        ! Point 20: (1430, 300) [work]
        CurrentX:=1430;
        CurrentY:=300;
        pCurrent.trans:=[-1*CurrentX,CurrentY,WorkZ];
        pCurrent.rot:=OrientZYX(0,0,180);
        pCurrent.robconf:=[1,0,-2,0];
        CalcTrack:=Bed1Wyong.uframe.trans.x+pCurrent.trans.x;
        IF CurrentY<1000 THEN CalcTrack:=CalcTrack+1200; ENDIF
        IF CalcTrack<TrackMin THEN CalcTrack:=TrackMin; ENDIF
        IF CalcTrack>TrackMax THEN CalcTrack:=TrackMax; ENDIF
        pCurrent.extax:=[CalcTrack,9E+09,9E+09,9E+09,9E+09,9E+09];
        MoveL pCurrent,vTravel,fine,tHeli\WObj:=Bed1Wyong;

        ! Point 21: (1730, 300) [work]
        CurrentX:=1730;
        CurrentY:=300;
        pCurrent.trans:=[-1*CurrentX,CurrentY,WorkZ];
        pCurrent.rot:=OrientZYX(0,0,180);
        pCurrent.robconf:=[1,0,-2,0];
        CalcTrack:=Bed1Wyong.uframe.trans.x+pCurrent.trans.x;
        IF CurrentY<1000 THEN CalcTrack:=CalcTrack+1200; ENDIF
        IF CalcTrack<TrackMin THEN CalcTrack:=TrackMin; ENDIF
        IF CalcTrack>TrackMax THEN CalcTrack:=TrackMax; ENDIF
        pCurrent.extax:=[CalcTrack,9E+09,9E+09,9E+09,9E+09,9E+09];
        MoveL pCurrent,vTravel,fine,tHeli\WObj:=Bed1Wyong;

        ! Point 22: (1730, 1550) [work]
        CurrentX:=1730;
        CurrentY:=1550;
        pCurrent.trans:=[-1*CurrentX,CurrentY,WorkZ];
        pCurrent.rot:=OrientZYX(0,0,180);
        pCurrent.robconf:=[1,0,-2,0];
        CalcTrack:=Bed1Wyong.uframe.trans.x+pCurrent.trans.x;
        IF CurrentY<1000 THEN CalcTrack:=CalcTrack+1200; ENDIF
        IF CalcTrack<TrackMin THEN CalcTrack:=TrackMin; ENDIF
        IF CalcTrack>TrackMax THEN CalcTrack:=TrackMax; ENDIF
        pCurrent.extax:=[CalcTrack,9E+09,9E+09,9E+09,9E+09,9E+09];
        MoveL pCurrent,vTravel,fine,tHeli\WObj:=Bed1Wyong;

        ! Point 23: (2030, 1550) [work]
        CurrentX:=2030;
        CurrentY:=1550;
        pCurrent.trans:=[-1*CurrentX,CurrentY,WorkZ];
        pCurrent.rot:=OrientZYX(0,0,180);
        pCurrent.robconf:=[1,0,-2,0];
        CalcTrack:=Bed1Wyong.uframe.trans.x+pCurrent.trans.x;
        IF CurrentY<1000 THEN CalcTrack:=CalcTrack+1200; ENDIF
        IF CalcTrack<TrackMin THEN CalcTrack:=TrackMin; ENDIF
        IF CalcTrack>TrackMax THEN CalcTrack:=TrackMax; ENDIF
        pCurrent.extax:=[CalcTrack,9E+09,9E+09,9E+09,9E+09,9E+09];
        MoveL pCurrent,vTravel,fine,tHeli\WObj:=Bed1Wyong;

        ! Point 24: (2030, 300) [work]
        CurrentX:=2030;
        CurrentY:=300;
        pCurrent.trans:=[-1*CurrentX,CurrentY,WorkZ];
        pCurrent.rot:=OrientZYX(0,0,180);
        pCurrent.robconf:=[1,0,-2,0];
        CalcTrack:=Bed1Wyong.uframe.trans.x+pCurrent.trans.x;
        IF CurrentY<1000 THEN CalcTrack:=CalcTrack+1200; ENDIF
        IF CalcTrack<TrackMin THEN CalcTrack:=TrackMin; ENDIF
        IF CalcTrack>TrackMax THEN CalcTrack:=TrackMax; ENDIF
        pCurrent.extax:=[CalcTrack,9E+09,9E+09,9E+09,9E+09,9E+09];
        MoveL pCurrent,vTravel,fine,tHeli\WObj:=Bed1Wyong;

        ! Point 25: (2330, 300) [work]
        CurrentX:=2330;
        CurrentY:=300;
        pCurrent.trans:=[-1*CurrentX,CurrentY,WorkZ];
        pCurrent.rot:=OrientZYX(0,0,180);
        pCurrent.robconf:=[1,0,-2,0];
        CalcTrack:=Bed1Wyong.uframe.trans.x+pCurrent.trans.x;
        IF CurrentY<1000 THEN CalcTrack:=CalcTrack+1200; ENDIF
        IF CalcTrack<TrackMin THEN CalcTrack:=TrackMin; ENDIF
        IF CalcTrack>TrackMax THEN CalcTrack:=TrackMax; ENDIF
        pCurrent.extax:=[CalcTrack,9E+09,9E+09,9E+09,9E+09,9E+09];
        MoveL pCurrent,vTravel,fine,tHeli\WObj:=Bed1Wyong;

        ! Point 26: (2330, 1550) [work]
        CurrentX:=2330;
        CurrentY:=1550;
        pCurrent.trans:=[-1*CurrentX,CurrentY,WorkZ];
        pCurrent.rot:=OrientZYX(0,0,180);
        pCurrent.robconf:=[1,0,-2,0];
        CalcTrack:=Bed1Wyong.uframe.trans.x+pCurrent.trans.x;
        IF CurrentY<1000 THEN CalcTrack:=CalcTrack+1200; ENDIF
        IF CalcTrack<TrackMin THEN CalcTrack:=TrackMin; ENDIF
        IF CalcTrack>TrackMax THEN CalcTrack:=TrackMax; ENDIF
        pCurrent.extax:=[CalcTrack,9E+09,9E+09,9E+09,9E+09,9E+09];
        MoveL pCurrent,vTravel,fine,tHeli\WObj:=Bed1Wyong;

        ! Point 27: (2630, 1550) [work]
        CurrentX:=2630;
        CurrentY:=1550;
        pCurrent.trans:=[-1*CurrentX,CurrentY,WorkZ];
        pCurrent.rot:=OrientZYX(0,0,180);
        pCurrent.robconf:=[1,0,-2,0];
        CalcTrack:=Bed1Wyong.uframe.trans.x+pCurrent.trans.x;
        IF CurrentY<1000 THEN CalcTrack:=CalcTrack+1200; ENDIF
        IF CalcTrack<TrackMin THEN CalcTrack:=TrackMin; ENDIF
        IF CalcTrack>TrackMax THEN CalcTrack:=TrackMax; ENDIF
        pCurrent.extax:=[CalcTrack,9E+09,9E+09,9E+09,9E+09,9E+09];
        MoveL pCurrent,vTravel,fine,tHeli\WObj:=Bed1Wyong;

        ! Point 28: (2630, 300) [work]
        CurrentX:=2630;
        CurrentY:=300;
        pCurrent.trans:=[-1*CurrentX,CurrentY,WorkZ];
        pCurrent.rot:=OrientZYX(0,0,180);
        pCurrent.robconf:=[1,0,-2,0];
        CalcTrack:=Bed1Wyong.uframe.trans.x+pCurrent.trans.x;
        IF CurrentY<1000 THEN CalcTrack:=CalcTrack+1200; ENDIF
        IF CalcTrack<TrackMin THEN CalcTrack:=TrackMin; ENDIF
        IF CalcTrack>TrackMax THEN CalcTrack:=TrackMax; ENDIF
        pCurrent.extax:=[CalcTrack,9E+09,9E+09,9E+09,9E+09,9E+09];
        MoveL pCurrent,vTravel,fine,tHeli\WObj:=Bed1Wyong;

        ! Point 29: (2930, 300) [work]
        CurrentX:=2930;
        CurrentY:=300;
        pCurrent.trans:=[-1*CurrentX,CurrentY,WorkZ];
        pCurrent.rot:=OrientZYX(0,0,180);
        pCurrent.robconf:=[1,0,-2,0];
        CalcTrack:=Bed1Wyong.uframe.trans.x+pCurrent.trans.x;
        IF CurrentY<1000 THEN CalcTrack:=CalcTrack+1200; ENDIF
        IF CalcTrack<TrackMin THEN CalcTrack:=TrackMin; ENDIF
        IF CalcTrack>TrackMax THEN CalcTrack:=TrackMax; ENDIF
        pCurrent.extax:=[CalcTrack,9E+09,9E+09,9E+09,9E+09,9E+09];
        MoveL pCurrent,vTravel,fine,tHeli\WObj:=Bed1Wyong;

        ! Point 30: (2930, 1550) [work]
        CurrentX:=2930;
        CurrentY:=1550;
        pCurrent.trans:=[-1*CurrentX,CurrentY,WorkZ];
        pCurrent.rot:=OrientZYX(0,0,180);
        pCurrent.robconf:=[1,0,-2,0];
        CalcTrack:=Bed1Wyong.uframe.trans.x+pCurrent.trans.x;
        IF CurrentY<1000 THEN CalcTrack:=CalcTrack+1200; ENDIF
        IF CalcTrack<TrackMin THEN CalcTrack:=TrackMin; ENDIF
        IF CalcTrack>TrackMax THEN CalcTrack:=TrackMax; ENDIF
        pCurrent.extax:=[CalcTrack,9E+09,9E+09,9E+09,9E+09,9E+09];
        MoveL pCurrent,vTravel,fine,tHeli\WObj:=Bed1Wyong;

        ! Point 31: (3230, 1550) [work]
        CurrentX:=3230;
        CurrentY:=1550;
        pCurrent.trans:=[-1*CurrentX,CurrentY,WorkZ];
        pCurrent.rot:=OrientZYX(0,0,180);
        pCurrent.robconf:=[1,0,-2,0];
        CalcTrack:=Bed1Wyong.uframe.trans.x+pCurrent.trans.x;
        IF CurrentY<1000 THEN CalcTrack:=CalcTrack+1200; ENDIF
        IF CalcTrack<TrackMin THEN CalcTrack:=TrackMin; ENDIF
        IF CalcTrack>TrackMax THEN CalcTrack:=TrackMax; ENDIF
        pCurrent.extax:=[CalcTrack,9E+09,9E+09,9E+09,9E+09,9E+09];
        MoveL pCurrent,vTravel,fine,tHeli\WObj:=Bed1Wyong;

        ! Point 32: (3230, 300) [work]
        CurrentX:=3230;
        CurrentY:=300;
        pCurrent.trans:=[-1*CurrentX,CurrentY,WorkZ];
        pCurrent.rot:=OrientZYX(0,0,180);
        pCurrent.robconf:=[1,0,-2,0];
        CalcTrack:=Bed1Wyong.uframe.trans.x+pCurrent.trans.x;
        IF CurrentY<1000 THEN CalcTrack:=CalcTrack+1200; ENDIF
        IF CalcTrack<TrackMin THEN CalcTrack:=TrackMin; ENDIF
        IF CalcTrack>TrackMax THEN CalcTrack:=TrackMax; ENDIF
        pCurrent.extax:=[CalcTrack,9E+09,9E+09,9E+09,9E+09,9E+09];
        MoveL pCurrent,vTravel,fine,tHeli\WObj:=Bed1Wyong;

        ! Point 33: (3530, 300) [work]
        CurrentX:=3530;
        CurrentY:=300;
        pCurrent.trans:=[-1*CurrentX,CurrentY,WorkZ];
        pCurrent.rot:=OrientZYX(0,0,180);
        pCurrent.robconf:=[1,0,-2,0];
        CalcTrack:=Bed1Wyong.uframe.trans.x+pCurrent.trans.x;
        IF CurrentY<1000 THEN CalcTrack:=CalcTrack+1200; ENDIF
        IF CalcTrack<TrackMin THEN CalcTrack:=TrackMin; ENDIF
        IF CalcTrack>TrackMax THEN CalcTrack:=TrackMax; ENDIF
        pCurrent.extax:=[CalcTrack,9E+09,9E+09,9E+09,9E+09,9E+09];
        MoveL pCurrent,vTravel,fine,tHeli\WObj:=Bed1Wyong;

        ! Point 34: (3530, 1550) [work]
        CurrentX:=3530;
        CurrentY:=1550;
        pCurrent.trans:=[-1*CurrentX,CurrentY,WorkZ];
        pCurrent.rot:=OrientZYX(0,0,180);
        pCurrent.robconf:=[1,0,-2,0];
        CalcTrack:=Bed1Wyong.uframe.trans.x+pCurrent.trans.x;
        IF CurrentY<1000 THEN CalcTrack:=CalcTrack+1200; ENDIF
        IF CalcTrack<TrackMin THEN CalcTrack:=TrackMin; ENDIF
        IF CalcTrack>TrackMax THEN CalcTrack:=TrackMax; ENDIF
        pCurrent.extax:=[CalcTrack,9E+09,9E+09,9E+09,9E+09,9E+09];
        MoveL pCurrent,vTravel,fine,tHeli\WObj:=Bed1Wyong;

        ! Point 35: (3830, 1550) [work]
        CurrentX:=3830;
        CurrentY:=1550;
        pCurrent.trans:=[-1*CurrentX,CurrentY,WorkZ];
        pCurrent.rot:=OrientZYX(0,0,180);
        pCurrent.robconf:=[1,0,-2,0];
        CalcTrack:=Bed1Wyong.uframe.trans.x+pCurrent.trans.x;
        IF CurrentY<1000 THEN CalcTrack:=CalcTrack+1200; ENDIF
        IF CalcTrack<TrackMin THEN CalcTrack:=TrackMin; ENDIF
        IF CalcTrack>TrackMax THEN CalcTrack:=TrackMax; ENDIF
        pCurrent.extax:=[CalcTrack,9E+09,9E+09,9E+09,9E+09,9E+09];
        MoveL pCurrent,vTravel,fine,tHeli\WObj:=Bed1Wyong;

        ! Point 36: (3830, 300) [work]
        CurrentX:=3830;
        CurrentY:=300;
        pCurrent.trans:=[-1*CurrentX,CurrentY,WorkZ];
        pCurrent.rot:=OrientZYX(0,0,180);
        pCurrent.robconf:=[1,0,-2,0];
        CalcTrack:=Bed1Wyong.uframe.trans.x+pCurrent.trans.x;
        IF CurrentY<1000 THEN CalcTrack:=CalcTrack+1200; ENDIF
        IF CalcTrack<TrackMin THEN CalcTrack:=TrackMin; ENDIF
        IF CalcTrack>TrackMax THEN CalcTrack:=TrackMax; ENDIF
        pCurrent.extax:=[CalcTrack,9E+09,9E+09,9E+09,9E+09,9E+09];
        MoveL pCurrent,vTravel,fine,tHeli\WObj:=Bed1Wyong;

        ! Point 37: (4130, 300) [work]
        CurrentX:=4130;
        CurrentY:=300;
        pCurrent.trans:=[-1*CurrentX,CurrentY,WorkZ];
        pCurrent.rot:=OrientZYX(0,0,180);
        pCurrent.robconf:=[1,0,-2,0];
        CalcTrack:=Bed1Wyong.uframe.trans.x+pCurrent.trans.x;
        IF CurrentY<1000 THEN CalcTrack:=CalcTrack+1200; ENDIF
        IF CalcTrack<TrackMin THEN CalcTrack:=TrackMin; ENDIF
        IF CalcTrack>TrackMax THEN CalcTrack:=TrackMax; ENDIF
        pCurrent.extax:=[CalcTrack,9E+09,9E+09,9E+09,9E+09,9E+09];
        MoveL pCurrent,vTravel,fine,tHeli\WObj:=Bed1Wyong;

        ! Point 38: (4130, 1550) [work]
        CurrentX:=4130;
        CurrentY:=1550;
        pCurrent.trans:=[-1*CurrentX,CurrentY,WorkZ];
        pCurrent.rot:=OrientZYX(0,0,180);
        pCurrent.robconf:=[1,0,-2,0];
        CalcTrack:=Bed1Wyong.uframe.trans.x+pCurrent.trans.x;
        IF CurrentY<1000 THEN CalcTrack:=CalcTrack+1200; ENDIF
        IF CalcTrack<TrackMin THEN CalcTrack:=TrackMin; ENDIF
        IF CalcTrack>TrackMax THEN CalcTrack:=TrackMax; ENDIF
        pCurrent.extax:=[CalcTrack,9E+09,9E+09,9E+09,9E+09,9E+09];
        MoveL pCurrent,vTravel,fine,tHeli\WObj:=Bed1Wyong;

        ! Point 39: (4430, 1550) [work]
        CurrentX:=4430;
        CurrentY:=1550;
        pCurrent.trans:=[-1*CurrentX,CurrentY,WorkZ];
        pCurrent.rot:=OrientZYX(0,0,180);
        pCurrent.robconf:=[1,0,-2,0];
        CalcTrack:=Bed1Wyong.uframe.trans.x+pCurrent.trans.x;
        IF CurrentY<1000 THEN CalcTrack:=CalcTrack+1200; ENDIF
        IF CalcTrack<TrackMin THEN CalcTrack:=TrackMin; ENDIF
        IF CalcTrack>TrackMax THEN CalcTrack:=TrackMax; ENDIF
        pCurrent.extax:=[CalcTrack,9E+09,9E+09,9E+09,9E+09,9E+09];
        MoveL pCurrent,vTravel,fine,tHeli\WObj:=Bed1Wyong;

        ! Point 40: (4430, 300) [work]
        CurrentX:=4430;
        CurrentY:=300;
        pCurrent.trans:=[-1*CurrentX,CurrentY,WorkZ];
        pCurrent.rot:=OrientZYX(0,0,180);
        pCurrent.robconf:=[1,0,-2,0];
        CalcTrack:=Bed1Wyong.uframe.trans.x+pCurrent.trans.x;
        IF CurrentY<1000 THEN CalcTrack:=CalcTrack+1200; ENDIF
        IF CalcTrack<TrackMin THEN CalcTrack:=TrackMin; ENDIF
        IF CalcTrack>TrackMax THEN CalcTrack:=TrackMax; ENDIF
        pCurrent.extax:=[CalcTrack,9E+09,9E+09,9E+09,9E+09,9E+09];
        MoveL pCurrent,vTravel,fine,tHeli\WObj:=Bed1Wyong;

        ! Point 41: (4730, 300) [work]
        CurrentX:=4730;
        CurrentY:=300;
        pCurrent.trans:=[-1*CurrentX,CurrentY,WorkZ];
        pCurrent.rot:=OrientZYX(0,0,180);
        pCurrent.robconf:=[1,0,-2,0];
        CalcTrack:=Bed1Wyong.uframe.trans.x+pCurrent.trans.x;
        IF CurrentY<1000 THEN CalcTrack:=CalcTrack+1200; ENDIF
        IF CalcTrack<TrackMin THEN CalcTrack:=TrackMin; ENDIF
        IF CalcTrack>TrackMax THEN CalcTrack:=TrackMax; ENDIF
        pCurrent.extax:=[CalcTrack,9E+09,9E+09,9E+09,9E+09,9E+09];
        MoveL pCurrent,vTravel,fine,tHeli\WObj:=Bed1Wyong;

        ! Point 42: (4730, 1550) [work]
        CurrentX:=4730;
        CurrentY:=1550;
        pCurrent.trans:=[-1*CurrentX,CurrentY,WorkZ];
        pCurrent.rot:=OrientZYX(0,0,180);
        pCurrent.robconf:=[1,0,-2,0];
        CalcTrack:=Bed1Wyong.uframe.trans.x+pCurrent.trans.x;
        IF CurrentY<1000 THEN CalcTrack:=CalcTrack+1200; ENDIF
        IF CalcTrack<TrackMin THEN CalcTrack:=TrackMin; ENDIF
        IF CalcTrack>TrackMax THEN CalcTrack:=TrackMax; ENDIF
        pCurrent.extax:=[CalcTrack,9E+09,9E+09,9E+09,9E+09,9E+09];
        MoveL pCurrent,vTravel,fine,tHeli\WObj:=Bed1Wyong;

        ! Point 43: (5030, 1550) [work]
        CurrentX:=5030;
        CurrentY:=1550;
        pCurrent.trans:=[-1*CurrentX,CurrentY,WorkZ];
        pCurrent.rot:=OrientZYX(0,0,180);
        pCurrent.robconf:=[1,0,-2,0];
        CalcTrack:=Bed1Wyong.uframe.trans.x+pCurrent.trans.x;
        IF CurrentY<1000 THEN CalcTrack:=CalcTrack+1200; ENDIF
        IF CalcTrack<TrackMin THEN CalcTrack:=TrackMin; ENDIF
        IF CalcTrack>TrackMax THEN CalcTrack:=TrackMax; ENDIF
        pCurrent.extax:=[CalcTrack,9E+09,9E+09,9E+09,9E+09,9E+09];
        MoveL pCurrent,vTravel,fine,tHeli\WObj:=Bed1Wyong;

        ! Point 44: (5030, 300) [work]
        CurrentX:=5030;
        CurrentY:=300;
        pCurrent.trans:=[-1*CurrentX,CurrentY,WorkZ];
        pCurrent.rot:=OrientZYX(0,0,180);
        pCurrent.robconf:=[1,0,-2,0];
        CalcTrack:=Bed1Wyong.uframe.trans.x+pCurrent.trans.x;
        IF CurrentY<1000 THEN CalcTrack:=CalcTrack+1200; ENDIF
        IF CalcTrack<TrackMin THEN CalcTrack:=TrackMin; ENDIF
        IF CalcTrack>TrackMax THEN CalcTrack:=TrackMax; ENDIF
        pCurrent.extax:=[CalcTrack,9E+09,9E+09,9E+09,9E+09,9E+09];
        MoveL pCurrent,vTravel,fine,tHeli\WObj:=Bed1Wyong;

        ! Point 45: (5330, 300) [work]
        CurrentX:=5330;
        CurrentY:=300;
        pCurrent.trans:=[-1*CurrentX,CurrentY,WorkZ];
        pCurrent.rot:=OrientZYX(0,0,180);
        pCurrent.robconf:=[1,0,-2,0];
        CalcTrack:=Bed1Wyong.uframe.trans.x+pCurrent.trans.x;
        IF CurrentY<1000 THEN CalcTrack:=CalcTrack+1200; ENDIF
        IF CalcTrack<TrackMin THEN CalcTrack:=TrackMin; ENDIF
        IF CalcTrack>TrackMax THEN CalcTrack:=TrackMax; ENDIF
        pCurrent.extax:=[CalcTrack,9E+09,9E+09,9E+09,9E+09,9E+09];
        MoveL pCurrent,vTravel,fine,tHeli\WObj:=Bed1Wyong;

        ! Point 46: (5330, 1550) [work]
        CurrentX:=5330;
        CurrentY:=1550;
        pCurrent.trans:=[-1*CurrentX,CurrentY,WorkZ];
        pCurrent.rot:=OrientZYX(0,0,180);
        pCurrent.robconf:=[1,0,-2,0];
        CalcTrack:=Bed1Wyong.uframe.trans.x+pCurrent.trans.x;
        IF CurrentY<1000 THEN CalcTrack:=CalcTrack+1200; ENDIF
        IF CalcTrack<TrackMin THEN CalcTrack:=TrackMin; ENDIF
        IF CalcTrack>TrackMax THEN CalcTrack:=TrackMax; ENDIF
        pCurrent.extax:=[CalcTrack,9E+09,9E+09,9E+09,9E+09,9E+09];
        MoveL pCurrent,vTravel,fine,tHeli\WObj:=Bed1Wyong;

        ! Point 47: (5630, 1550) [work]
        CurrentX:=5630;
        CurrentY:=1550;
        pCurrent.trans:=[-1*CurrentX,CurrentY,WorkZ];
        pCurrent.rot:=OrientZYX(0,0,180);
        pCurrent.robconf:=[1,0,-2,0];
        CalcTrack:=Bed1Wyong.uframe.trans.x+pCurrent.trans.x;
        IF CurrentY<1000 THEN CalcTrack:=CalcTrack+1200; ENDIF
        IF CalcTrack<TrackMin THEN CalcTrack:=TrackMin; ENDIF
        IF CalcTrack>TrackMax THEN CalcTrack:=TrackMax; ENDIF
        pCurrent.extax:=[CalcTrack,9E+09,9E+09,9E+09,9E+09,9E+09];
        MoveL pCurrent,vTravel,fine,tHeli\WObj:=Bed1Wyong;

        ! Point 48: (5630, 300) [work]
        CurrentX:=5630;
        CurrentY:=300;
        pCurrent.trans:=[-1*CurrentX,CurrentY,WorkZ];
        pCurrent.rot:=OrientZYX(0,0,180);
        pCurrent.robconf:=[1,0,-2,0];
        CalcTrack:=Bed1Wyong.uframe.trans.x+pCurrent.trans.x;
        IF CurrentY<1000 THEN CalcTrack:=CalcTrack+1200; ENDIF
        IF CalcTrack<TrackMin THEN CalcTrack:=TrackMin; ENDIF
        IF CalcTrack>TrackMax THEN CalcTrack:=TrackMax; ENDIF
        pCurrent.extax:=[CalcTrack,9E+09,9E+09,9E+09,9E+09,9E+09];
        MoveL pCurrent,vTravel,fine,tHeli\WObj:=Bed1Wyong;

        ! Point 49: (5930, 300) [work]
        CurrentX:=5930;
        CurrentY:=300;
        pCurrent.trans:=[-1*CurrentX,CurrentY,WorkZ];
        pCurrent.rot:=OrientZYX(0,0,180);
        pCurrent.robconf:=[1,0,-2,0];
        CalcTrack:=Bed1Wyong.uframe.trans.x+pCurrent.trans.x;
        IF CurrentY<1000 THEN CalcTrack:=CalcTrack+1200; ENDIF
        IF CalcTrack<TrackMin THEN CalcTrack:=TrackMin; ENDIF
        IF CalcTrack>TrackMax THEN CalcTrack:=TrackMax; ENDIF
        pCurrent.extax:=[CalcTrack,9E+09,9E+09,9E+09,9E+09,9E+09];
        MoveL pCurrent,vTravel,fine,tHeli\WObj:=Bed1Wyong;

        ! Point 50: (5930, 1550) [work]
        CurrentX:=5930;
        CurrentY:=1550;
        pCurrent.trans:=[-1*CurrentX,CurrentY,WorkZ];
        pCurrent.rot:=OrientZYX(0,0,180);
        pCurrent.robconf:=[1,0,-2,0];
        CalcTrack:=Bed1Wyong.uframe.trans.x+pCurrent.trans.x;
        IF CurrentY<1000 THEN CalcTrack:=CalcTrack+1200; ENDIF
        IF CalcTrack<TrackMin THEN CalcTrack:=TrackMin; ENDIF
        IF CalcTrack>TrackMax THEN CalcTrack:=TrackMax; ENDIF
        pCurrent.extax:=[CalcTrack,9E+09,9E+09,9E+09,9E+09,9E+09];
        MoveL pCurrent,vTravel,fine,tHeli\WObj:=Bed1Wyong;

        ! Stop blade rotation
        HeliBladeSpeed 0,"FWD";
        WaitTime 1;

        ! Lift to safe height
        CurrentJoints:=CJointT();
        CurrentPos:=CalcRobT(CurrentJoints,tHeli\WObj:=Bed1Wyong);
        MoveL Offs(CurrentPos,0,0,200),v200,z5,tHeli\WObj:=Bed1Wyong;

        ! Return tool and go home
        TPWrite "Py2Pan: Dropping off helicopter...";
        Heli_Dropoff;
        Home FALSE;

        TPWrite "========================================";
        TPWrite "Py2Pan: COMPLETE";
        TPWrite "========================================";

    ERROR
        HeliBladeSpeed 0,"FWD";
        IF bFCActive THEN
            FCPressEnd Offs(CurrentPos,0,0,100),v50,\DeactOnly,tHeli\WObj:=Bed1Wyong;
        ENDIF
        RAISE;
    ENDPROC

    PROC Py2VS()
        ! Py2VS - Generated by Onyx Tool Class
        ! Workzone: panel
        ! Area: (580,350) to (5880,1500)
        ! Z = 455mm
        ! Step: 200mm

        VAR robtarget pCurrent;
        VAR jointtarget CurrentJoints;
        VAR robtarget CurrentPos;
        VAR num WorkZ:=455;
        VAR num SafeZ:=655;
        VAR num CurrentX:=0;
        VAR num CurrentY:=0;
        VAR speeddata vTravel:=[75,15,2000,15];
        VAR num TrackMin:=-300;
        VAR num TrackMax:=10050;
        VAR num CalcTrack:=0;

        TPWrite "========================================";
        TPWrite "Py2VS: Starting";
        TPWrite "========================================";
        TPWrite "Workzone: panel";
        TPWrite "WorkZ=" \Num:=WorkZ;

        ! Get tool if needed
        UpdateToolNum;
        IF ToolNum<>3 THEN
            TPWrite "Py2VS: Getting tool...";
            Home TRUE;
            VS_Pickup;
        ELSE
            CurrentJoints:=CJointT();
            CurrentPos:=CalcRobT(CurrentJoints,tVS\WObj:=wobj0);
            IF (CurrentPos.trans.x)>8000 AND CurrentPos.trans.z<400 THEN
                MoveL Offs(CurrentPos,0,0,(400-CurrentPos.trans.z)),v100,z5,tVS;
            ENDIF
        ENDIF

        ! ========================================
        ! Pattern Execution: 4 points
        ! Force Monitoring: DISABLED
        ! ========================================

        ! Use VS tool's orientation from pickup end position (pVSHome3)
        ! This prevents 180 degree rotation when moving to work surface
        pCurrent.rot:=pVSHome3.rot;

        ! Point 1: (173, 1850) [rapid]
        CurrentX:=173;
        CurrentY:=1850;
        pCurrent.trans:=[-1*CurrentX,CurrentY,SafeZ];
        pCurrent.robconf:=[1,0,1,0];
        CalcTrack:=Bed1Wyong.uframe.trans.x+pCurrent.trans.x;
        IF CurrentY<1000 THEN CalcTrack:=CalcTrack+1200; ENDIF
        IF CalcTrack<TrackMin THEN CalcTrack:=TrackMin; ENDIF
        IF CalcTrack>TrackMax THEN CalcTrack:=TrackMax; ENDIF
        pCurrent.extax:=[CalcTrack,9E+09,9E+09,9E+09,9E+09,9E+09];
        MoveJ pCurrent,v500,z5,tVS\WObj:=Bed1Wyong;

        ! Turn on vibrating screed after positioning
        TPWrite "Py2VS: Starting screed...";
        VS_on;

        ! Point 2: (223, 1850) [work]
        CurrentX:=223;
        CurrentY:=1850;
        pCurrent.trans:=[-1*CurrentX,CurrentY,WorkZ];
        pCurrent.robconf:=[1,0,1,0];
        CalcTrack:=Bed1Wyong.uframe.trans.x+pCurrent.trans.x;
        IF CurrentY<1000 THEN CalcTrack:=CalcTrack+1200; ENDIF
        IF CalcTrack<TrackMin THEN CalcTrack:=TrackMin; ENDIF
        IF CalcTrack>TrackMax THEN CalcTrack:=TrackMax; ENDIF
        pCurrent.extax:=[CalcTrack,9E+09,9E+09,9E+09,9E+09,9E+09];
        MoveL pCurrent,vTravel,fine,tVS\WObj:=Bed1Wyong;

        ! Point 3: (6237, 1850) [work]
        CurrentX:=6237;
        CurrentY:=1850;
        pCurrent.trans:=[-1*CurrentX,CurrentY,WorkZ];
        pCurrent.robconf:=[1,0,1,0];
        CalcTrack:=Bed1Wyong.uframe.trans.x+pCurrent.trans.x;
        IF CurrentY<1000 THEN CalcTrack:=CalcTrack+1200; ENDIF
        IF CalcTrack<TrackMin THEN CalcTrack:=TrackMin; ENDIF
        IF CalcTrack>TrackMax THEN CalcTrack:=TrackMax; ENDIF
        pCurrent.extax:=[CalcTrack,9E+09,9E+09,9E+09,9E+09,9E+09];
        MoveL pCurrent,vTravel,fine,tVS\WObj:=Bed1Wyong;

        ! Point 4: (6287, 1850) [rapid]
        CurrentX:=6287;
        CurrentY:=1850;
        pCurrent.trans:=[-1*CurrentX,CurrentY,SafeZ];
        pCurrent.robconf:=[1,0,1,0];
        CalcTrack:=Bed1Wyong.uframe.trans.x+pCurrent.trans.x;
        IF CurrentY<1000 THEN CalcTrack:=CalcTrack+1200; ENDIF
        IF CalcTrack<TrackMin THEN CalcTrack:=TrackMin; ENDIF
        IF CalcTrack>TrackMax THEN CalcTrack:=TrackMax; ENDIF
        pCurrent.extax:=[CalcTrack,9E+09,9E+09,9E+09,9E+09,9E+09];
        MoveJ pCurrent,v500,z5,tVS\WObj:=Bed1Wyong;

        VS_off;

        ! Lift to safe height
        CurrentJoints:=CJointT();
        CurrentPos:=CalcRobT(CurrentJoints,tVS\WObj:=Bed1Wyong);
        MoveL Offs(CurrentPos,0,0,200),v200,z5,tVS\WObj:=Bed1Wyong;

        ! Return tool and go home
        TPWrite "Py2VS: Dropping off tool...";
        VS_Dropoff;
        Home FALSE;

        TPWrite "========================================";
        TPWrite "Py2VS: COMPLETE";
        TPWrite "========================================";

    ERROR
        VS_off;
        TPWrite "Py2VS ERROR: " \Num:=ERRNO;
        RAISE;
    ENDPROC


    PROC SeqBedClean()
        ! SeqBedClean - Bed Cleaning Sequence
        ! Runs: Vacuum -> Polish
        ! Generated by Onyx Toolpath Generator v2

        TPWrite "========================================";
        TPWrite "SeqBedClean: Starting Bed Clean Sequence";
        TPWrite "========================================";
        TPWrite "Step 1: Vacuum";
        TPWrite "Step 2: Polish";
        TPWrite "========================================";

        ! Step 1: Vacuum the bed
        TPWrite "SeqBedClean: Starting vacuum...";
        Py2Vac;
        TPWrite "SeqBedClean: Vacuum complete";

        ! Step 2: Polish the bed
        TPWrite "SeqBedClean: Starting polish...";
        Py2Polish;
        TPWrite "SeqBedClean: Polish complete";

        TPWrite "========================================";
        TPWrite "SeqBedClean: SEQUENCE COMPLETE";
        TPWrite "========================================";

    ERROR
        TPWrite "SeqBedClean ERROR: " \Num:=ERRNO;
        RAISE;
    ENDPROC


    ! ========== END PY2 GENERATED PROCEDURES ==========

ENDMODULE
